// TIA Portal project "S7-1200-Tank-Level-Control" (V17)

(* hardware
DEVICE "S7-1200 station_1"  S7-1200 Station
   slot 0: "Rack_0"  S7-1200 Rack  Rack  V1.0
   slot 1: "PLC_1"  CPU 1212C DC/DC/DC  6ES7 212-1AE40-0XB0  V4.2
DEVICE "HMI_1"  TP700 Comfort
   slot 0: "HMI_1"  TP700 Comfort  6AV2 124-0GC01-0AX0  17.0.0.0
   slot 1: "HMI_RT_1"  TP700 Comfort  6AV2 124-0GC01-0AX0  17.0.0.0
   slot 5: "HMI_1.IE_CP_1"  PROFINET Interface  17.0.0.0
      slot 1: "PROFINET Interface_1"  PROFINET Interface
         slot 1: "Port_1"  Port
         slot 2: "Port_2"  Port
   slot 7: "HMI_1.MPI/DP_CP_1"  MPI/DP Interface  17.0.0.0
*)

// ===== PLC "PLC_1"  CPU 1212C DC/DC/DC =====

DATA_BLOCK "DB_Control"   // DB1
{ S7_Optimized_Access := 'TRUE' }
VERSION : 0.1
   VAR
      AutoMode : Bool;   // Automatic operating mode
      ManualInletCmd : Real;   // Manual inlet valve command [%]
      ManualOutletCmd : Real;   // Manual outlet valve command [%]
      PIDInletCmd : Real;   // PID controller output [%]
      InletValveCmd : Real;   // Final inlet valve command [%]
      OutletValveCmd : Real;   // Final outlet valve command [%]
      LevelSetpoint : Real := 50.0;   // Tank level setpoint [%]
      Level_H : Bool;   // High level alarm
      Level_HH : Bool;   // High-high level protection
      Level_L : Bool;   // Low level alarm
      Level_LL : Bool;   // Low-low level protection
      HMI_AlarmWord : Word;   // HMI alarm trigger word
      ManualPumpCmd : Bool;   // Manual pump command
      PumpManualControlEnable : Bool;   // Manual pump control permission
   END_VAR
BEGIN
END_DATA_BLOCK

DATA_BLOCK "DB_TankSimulation"   // DB2
{ S7_Optimized_Access := 'TRUE' }
VERSION : 0.1
// stored: InstanceOfName FB_TankSimulation
"FB_TankSimulation"
BEGIN
END_DATA_BLOCK

FUNCTION_BLOCK "FB_TankSimulation"   // FB1, SCL
{ S7_Optimized_Access := 'TRUE' }
VERSION : 0.1
   VAR_INPUT
      CycleTime : Real := 0.1;
      InletValveCmd : Real;
      OutletValveCmd : Real;
   END_VAR
   VAR
      TankLevel : Real;
      Inflow : Real;
      Outflow : Real;
      InletValveActual : Real;
      OutletValveActual : Real;
      ValveSpeed : Real := 5.0;
      PumpRunning : Bool;
      PumpSpeed : Real := 2.0;
      PumpTimer : Real;
      PumpFailureSimulation : Bool;
      PumpFault : Bool;
      PumpFaultReset : Bool;
      PumpCmd : Bool;
   END_VAR
BEGIN
   REGION Pump_simulation

       IF #PumpCmd AND NOT #PumpFault THEN
           #PumpTimer := #PumpTimer + (#PumpSpeed * #CycleTime);

           IF #PumpTimer >= 2.0 AND NOT #PumpFailureSimulation THEN
               #PumpRunning := TRUE;
               #PumpTimer := 2.0;

           ELSIF #PumpTimer >= 4.0 AND #PumpFailureSimulation THEN
               #PumpFault := TRUE;
               #PumpTimer := 0.0;
           END_IF;

       END_IF;

       IF NOT #PumpCmd THEN
           #PumpTimer := #PumpTimer - (#PumpSpeed * #CycleTime);

           IF #PumpTimer <= 0.0 THEN
               #PumpRunning := FALSE;
               #PumpTimer := 0.0;
           END_IF;

       END_IF;

       IF #PumpFailureSimulation AND #PumpRunning THEN
           #PumpRunning := FALSE;
           #PumpFault := TRUE;
           #PumpTimer := 0.0;
       END_IF;

       IF #PumpFaultReset AND NOT #PumpFailureSimulation THEN
           #PumpFault := FALSE;
       END_IF;

   END_REGION


   REGION Inlet_valve_simulation

       IF #InletValveActual < #InletValveCmd THEN
           #InletValveActual := #InletValveActual + (#ValveSpeed * #CycleTime);

           IF #InletValveActual > #InletValveCmd THEN
               #InletValveActual := #InletValveCmd;
           END_IF;

       ELSIF #InletValveActual > #InletValveCmd THEN
           #InletValveActual := #InletValveActual - (#ValveSpeed * #CycleTime);

           IF #InletValveActual < #InletValveCmd THEN
               #InletValveActual := #InletValveCmd;
           END_IF;

       END_IF;

   END_REGION


   REGION Outlet_valve_simulation

       IF #OutletValveActual < #OutletValveCmd THEN
           #OutletValveActual := #OutletValveActual + (#ValveSpeed * #CycleTime);

           IF #OutletValveActual > #OutletValveCmd THEN
               #OutletValveActual := #OutletValveCmd;
           END_IF;

       ELSIF #OutletValveActual > #OutletValveCmd THEN
           #OutletValveActual := #OutletValveActual - (#ValveSpeed * #CycleTime);

           IF #OutletValveActual < #OutletValveCmd THEN
               #OutletValveActual := #OutletValveCmd;
           END_IF;

       END_IF;

   END_REGION


   REGION Flow_calculation

       IF #PumpRunning THEN
           #Inflow := (#InletValveActual / 100.0) * 2.0;
       ELSE
           #Inflow := 0.0;
       END_IF;

       #Outflow := (#OutletValveActual / 100.0) * 2.0;

   END_REGION


   REGION Tank_level_simulation

       #TankLevel := #TankLevel + (#Inflow - #Outflow) * #CycleTime;

       IF #TankLevel > 100.0 THEN
           #TankLevel := 100.0;
       END_IF;

       IF #TankLevel < 0.0 THEN
           #TankLevel := 0.0;
       END_IF;

   END_REGION
END_FUNCTION_BLOCK

ORGANIZATION_BLOCK "Main"   // OB1, LAD, ProgramCycle
TITLE = "Main Program Sweep (Cycle)"
{ S7_Optimized_Access := 'TRUE' }
VERSION : 0.1
   VAR_INPUT
      Initial_Call : Bool;   // Initial call of this OB
      Remanence : Bool;   // =True, if remanent data are available
   END_VAR
BEGIN

REGION Network 1: Operating mode command selection
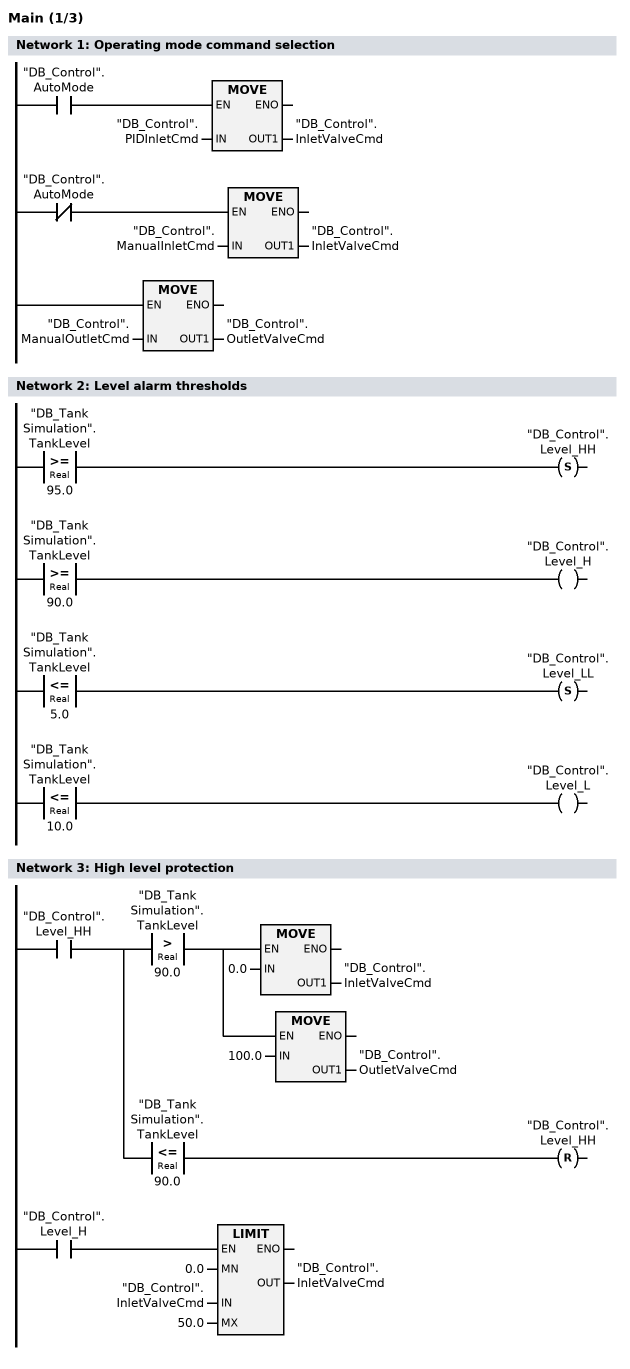
   RUNG wire#powerrail
      Contact( "DB_Control".AutoMode )
      Move(in := "DB_Control".PIDInletCmd, out1 => "DB_Control".InletValveCmd)
   END_RUNG
   RUNG wire#powerrail
      I_Contact( "DB_Control".AutoMode )
      Move(in := "DB_Control".ManualInletCmd, out1 => "DB_Control".InletValveCmd)
   END_RUNG
   RUNG wire#powerrail
      Move(in := "DB_Control".ManualOutletCmd, out1 => "DB_Control".OutletValveCmd)
   END_RUNG
   // the same network as SCL:
   IF "DB_Control".AutoMode THEN "DB_Control".InletValveCmd := "DB_Control".PIDInletCmd; END_IF;
   IF NOT "DB_Control".AutoMode THEN "DB_Control".InletValveCmd := "DB_Control".ManualInletCmd; END_IF;
   "DB_Control".OutletValveCmd := "DB_Control".ManualOutletCmd;
END_REGION

REGION Network 2: Level alarm thresholds
   RUNG wire#powerrail
      { S7_Templates := "SrcType := Real" } GE_Contact(in1 := "DB_TankSimulation".TankLevel, in2 := 95.0)
      S_Coil( "DB_Control".Level_HH )
   END_RUNG
   RUNG wire#powerrail
      { S7_Templates := "SrcType := Real" } GE_Contact(in1 := "DB_TankSimulation".TankLevel, in2 := 90.0)
      Coil( "DB_Control".Level_H )
   END_RUNG
   RUNG wire#powerrail
      { S7_Templates := "SrcType := Real" } LE_Contact(in1 := "DB_TankSimulation".TankLevel, in2 := 5.0)
      S_Coil( "DB_Control".Level_LL )
   END_RUNG
   RUNG wire#powerrail
      { S7_Templates := "SrcType := Real" } LE_Contact(in1 := "DB_TankSimulation".TankLevel, in2 := 10.0)
      Coil( "DB_Control".Level_L )
   END_RUNG
   // the same network as SCL:
   IF "DB_TankSimulation".TankLevel >= 95.0 THEN "DB_Control".Level_HH := TRUE; END_IF;
   "DB_Control".Level_H := "DB_TankSimulation".TankLevel >= 90.0;
   IF "DB_TankSimulation".TankLevel <= 5.0 THEN "DB_Control".Level_LL := TRUE; END_IF;
   "DB_Control".Level_L := "DB_TankSimulation".TankLevel <= 10.0;
END_REGION

REGION Network 3: High level protection
   IF "DB_Control".Level_HH AND ("DB_TankSimulation".TankLevel > 90.0) THEN
       "DB_Control".InletValveCmd := 0.0;
       "DB_Control".OutletValveCmd := 100.0;
   END_IF;
   IF "DB_Control".Level_HH AND ("DB_TankSimulation".TankLevel <= 90.0) THEN
       "DB_Control".Level_HH := FALSE;
   END_IF;
   IF "DB_Control".Level_H THEN
       "DB_Control".InletValveCmd := LIMIT(MN := 0.0, IN := "DB_Control".InletValveCmd, MX := 50.0);
   END_IF;
END_REGION

REGION Network 4: Low level protection
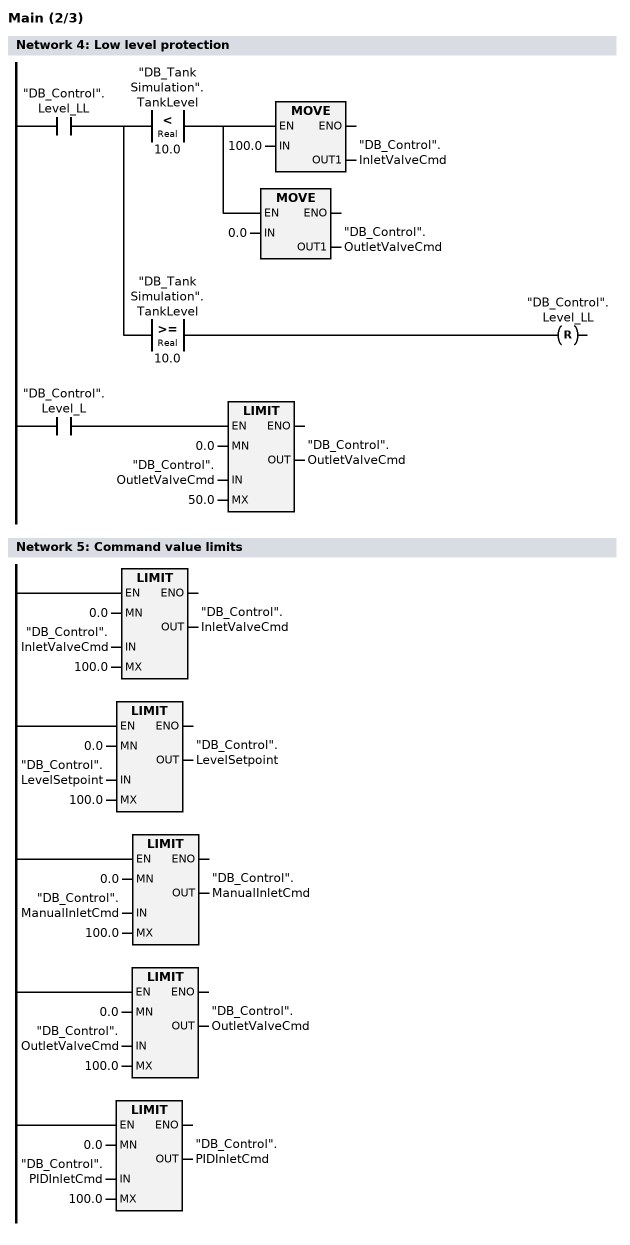
   IF "DB_Control".Level_LL AND ("DB_TankSimulation".TankLevel < 10.0) THEN
       "DB_Control".InletValveCmd := 100.0;
       "DB_Control".OutletValveCmd := 0.0;
   END_IF;
   IF "DB_Control".Level_LL AND ("DB_TankSimulation".TankLevel >= 10.0) THEN
       "DB_Control".Level_LL := FALSE;
   END_IF;
   IF "DB_Control".Level_L THEN
       "DB_Control".OutletValveCmd := LIMIT(MN := 0.0, IN := "DB_Control".OutletValveCmd, MX := 50.0);
   END_IF;
END_REGION

REGION Network 5: Command value limits
   "DB_Control".InletValveCmd := LIMIT(MN := 0.0, IN := "DB_Control".InletValveCmd, MX := 100.0);
   "DB_Control".LevelSetpoint := LIMIT(MN := 0.0, IN := "DB_Control".LevelSetpoint, MX := 100.0);
   "DB_Control".ManualInletCmd := LIMIT(MN := 0.0, IN := "DB_Control".ManualInletCmd, MX := 100.0);
   "DB_Control".OutletValveCmd := LIMIT(MN := 0.0, IN := "DB_Control".OutletValveCmd, MX := 100.0);
   "DB_Control".PIDInletCmd := LIMIT(MN := 0.0, IN := "DB_Control".PIDInletCmd, MX := 100.0);
END_REGION

REGION Network 6: HMI alarm word mapping
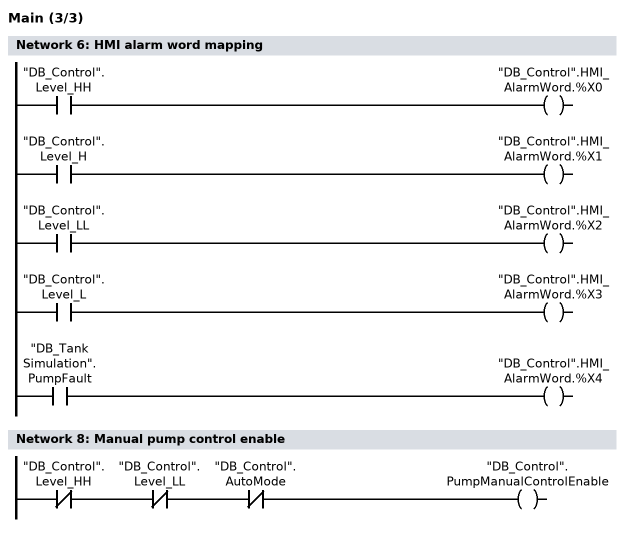
   RUNG wire#powerrail
      Contact( "DB_Control".Level_HH )
      Coil( "DB_Control".HMI_AlarmWord.%X0 )
   END_RUNG
   RUNG wire#powerrail
      Contact( "DB_Control".Level_H )
      Coil( "DB_Control".HMI_AlarmWord.%X1 )
   END_RUNG
   RUNG wire#powerrail
      Contact( "DB_Control".Level_LL )
      Coil( "DB_Control".HMI_AlarmWord.%X2 )
   END_RUNG
   RUNG wire#powerrail
      Contact( "DB_Control".Level_L )
      Coil( "DB_Control".HMI_AlarmWord.%X3 )
   END_RUNG
   RUNG wire#powerrail
      Contact( "DB_TankSimulation".PumpFault )
      Coil( "DB_Control".HMI_AlarmWord.%X4 )
   END_RUNG
   // the same network as SCL:
   "DB_Control".HMI_AlarmWord.%X0 := "DB_Control".Level_HH;
   "DB_Control".HMI_AlarmWord.%X1 := "DB_Control".Level_H;
   "DB_Control".HMI_AlarmWord.%X2 := "DB_Control".Level_LL;
   "DB_Control".HMI_AlarmWord.%X3 := "DB_Control".Level_L;
   "DB_Control".HMI_AlarmWord.%X4 := "DB_TankSimulation".PumpFault;
END_REGION

REGION Network 7 (SCL): Pump command control
   IF "DB_Control".Level_HH THEN
       "DB_TankSimulation".PumpCmd := FALSE;
   ELSIF "DB_Control".Level_LL THEN
       "DB_TankSimulation".PumpCmd := TRUE;
   ELSIF "DB_Control".AutoMode THEN
       "DB_TankSimulation".PumpCmd := TRUE;
   ELSE
       "DB_TankSimulation".PumpCmd := "DB_Control".ManualPumpCmd;

   END_IF;
END_REGION

REGION Network 8: Manual pump control enable
   RUNG wire#powerrail
      I_Contact( "DB_Control".Level_HH )
      I_Contact( "DB_Control".Level_LL )
      I_Contact( "DB_Control".AutoMode )
      Coil( "DB_Control".PumpManualControlEnable )
   END_RUNG
   // the same network as SCL:
   "DB_Control".PumpManualControlEnable := NOT "DB_Control".Level_HH AND NOT "DB_Control".Level_LL AND NOT "DB_Control".AutoMode;
END_REGION
END_ORGANIZATION_BLOCK

ORGANIZATION_BLOCK "OB_TankSimulation"   // OB30, LAD, CyclicInterrupt
{ S7_Optimized_Access := 'TRUE' }
VERSION : 0.1
   VAR_INPUT
      Initial_Call : Bool;   // Initial call of this OB
      Event_Count : Int;   // Events discarded
   END_VAR
BEGIN

REGION Network 1: Tank Simulation Execution
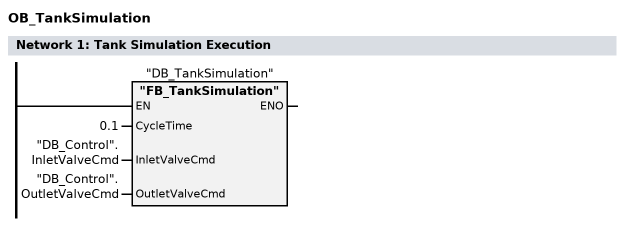
   RUNG wire#powerrail
      "DB_TankSimulation"(CycleTime := 0.1, InletValveCmd := "DB_Control".InletValveCmd, OutletValveCmd := "DB_Control".OutletValveCmd)
   END_RUNG
   // the same network as SCL:
   "DB_TankSimulation"(CycleTime := 0.1,   // "FB_TankSimulation"
                       InletValveCmd := "DB_Control".InletValveCmd,
                       OutletValveCmd := "DB_Control".OutletValveCmd);
END_REGION
END_ORGANIZATION_BLOCK

ORGANIZATION_BLOCK "OB_PID_Control"   // OB31, LAD, CyclicInterrupt
{ S7_Optimized_Access := 'TRUE' }
VERSION : 0.1
   VAR_INPUT
      Initial_Call : Bool;   // Initial call of this OB
      Event_Count : Int;   // Events discarded
   END_VAR
BEGIN

REGION Network 1: PID Controller Execution
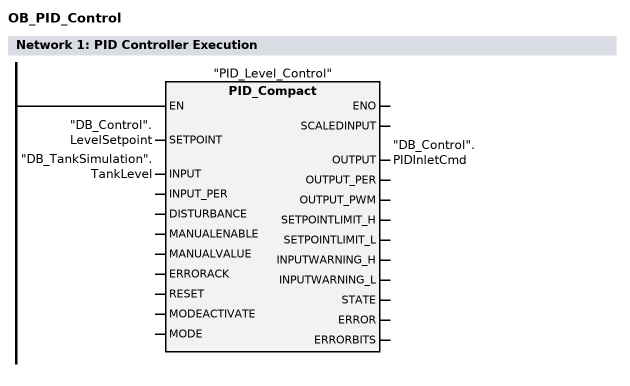
   "PID_Level_Control"(Setpoint := "DB_Control".LevelSetpoint,   // PID_Compact
                       Input := "DB_TankSimulation".TankLevel,
                       Output => "DB_Control".PIDInletCmd);
END_REGION
END_ORGANIZATION_BLOCK

(* ===== HMI "HMI_RT_1" =====
system functions are stored by id; their names below are inferred from use
connection "HMI_Connection_1": ETHERNET, S7_1200_OMS

HMI tags "Default tag table"
   "Tag_ScreenNumber" : UInt, internal
   "DB_Control_AutoMode" : Bool = PLC DB_Control.AutoMode, 1 s
   "DB_Control_LevelSetpoint" : Real = PLC DB_Control.LevelSetpoint, 1 s
   "DB_Control_ManualInletCmd" : Real = PLC DB_Control.ManualInletCmd, 1 s
   "DB_Control_OutletValveCmd" : Real = PLC DB_Control.OutletValveCmd, 1 s
   "DB_TankSimulation_TankLevel" : Real = PLC DB_TankSimulation.TankLevel, 1 s
   "DB_Control_PID_InletCmd" : Real = PLC DB_Control.PIDInletCmd, 1 s
   "DB_Control_InletValveCmd" : Real = PLC DB_Control.InletValveCmd, 1 s
   "DB_Control_Level_HH" : Bool = PLC DB_Control.Level_HH, 1 s
   "DB_Control_Level_H" : Bool = PLC DB_Control.Level_H, 1 s
   "DB_Control_Level_L" : Bool = PLC DB_Control.Level_L, 1 s
   "DB_Control_Level_LL" : Bool = PLC DB_Control.Level_LL, 1 s
   "DB_Control_ManualOutletCmd" : Real = PLC DB_Control.ManualOutletCmd, 1 s
   "DB_Control_HMI_AlarmWord" : Word = PLC DB_Control.HMI_AlarmWord, 1 s
   "DB_TankSimulation_OutletValveActual" : Real = PLC DB_TankSimulation.OutletValveActual, 1 s
   "DB_TankSimulation_InletValveActual" : Real = PLC DB_TankSimulation.InletValveActual, 1 s
   "DB_Control_ManualPumpCmd" : Bool = PLC DB_Control.ManualPumpCmd, 1 s
   "DB_TankSimulation_PumpRunning" : Bool = PLC DB_TankSimulation.PumpRunning, 1 s
   "DB_TankSimulation_PumpFault" : Bool = PLC DB_TankSimulation.PumpFault, 1 s
   "DB_TankSimulation_PumpFailureSimulation" : Bool = PLC DB_TankSimulation.PumpFailureSimulation, 1 s
   "DB_TankSimulation_PumpFaultReset" : Bool = PLC DB_TankSimulation.PumpFaultReset, 1 s
   "DB_Control_PumpManualControlEnable" : Bool = PLC DB_Control.PumpManualControlEnable, 1 s

discrete alarms
   1: 'Tank level above 95%', class Errors, trigger "DB_Control_HMI_AlarmWord" bit 0
   2: 'Tank level above 90%', class Warnings, trigger "DB_Control_HMI_AlarmWord" bit 1
   3: 'Tank level below 5%', class Errors, trigger "DB_Control_HMI_AlarmWord" bit 2
   4: 'Tank level below 10%', class Warnings, trigger "DB_Control_HMI_AlarmWord" bit 3
   5: 'Pump stopped', class Errors, trigger "DB_Control_HMI_AlarmWord" bit 4

screen "Tank Control" 800x428, template "Template_1"
   on GenerateScreen: SetTag("Tag_ScreenNumber", 1)
   TextField "Text field_1" at 89,0 size 149x23; Text 'CONTROL MODE'
   Circle "Circle_1" at 103,53 size 25x25
      Appearance <- "DB_Control_AutoMode"
   Circle "Circle_2" at 183,53 size 25x25
      Appearance <- "DB_Control_AutoMode"
   TextField "Text field_4" at 122,224 size 82x23; Text 'Setpoint'
   IOField "I/O field_1" at 128,247 size 67x32; FormatPattern 999
      ProcessValue <- "DB_Control_LevelSetpoint"
      ObjectEnable <- "DB_Control_AutoMode"
   TextField "Text field_5" at 163,251 size 25x23; Text '%'
   TextField "Text field_6" at 40,286 size 120x23; Text 'Manual Inlet'
   IOField "I/O field_2" at 62,308 size 67x32; FormatPattern 999
      ProcessValue <- "DB_Control_ManualInletCmd"
      ObjectEnable <- "DB_Control_AutoMode"
   TextField "Text field_7" at 97,312 size 25x23; Text '%'
   TextField "Text field_8" at 157,285 size 174x23; Text 'Outlet disturbance'
   IOField "I/O field_3" at 195,308 size 67x32; FormatPattern 999
      ProcessValue <- "DB_Control_ManualOutletCmd"
   TextField "Text field_9" at 230,312 size 25x23; Text '%'
   Bar "Bar_1" at 405,78 size 130x255; MinimumValue 0; MaximumValue 100
      ProcessValue <- "DB_TankSimulation_TankLevel"
   TextField "Text field_10" at 415,1 size 115x23; Text 'TANK LEVEL'
   IOField "I/O field_4" at 436,24 size 67x32; FormatPattern 999
      ProcessValue <- "DB_TankSimulation_TankLevel"
   TextField "Text field_11" at 471,28 size 25x23; Text '%'
   TextField "Text field_12" at 636,14 size 145x23; Text 'PROCESS DATA'
   TextField "Text field_13" at 611,47 size 82x23; Text 'Setpoint'
   IOField "I/O field_5" at 694,42 size 67x32; FormatPattern 999
      ProcessValue <- "DB_Control_LevelSetpoint"
   TextField "Text field_14" at 729,46 size 25x23; Text '%'
   TextField "Text field_15" at 611,85 size 104x23; Text 'Tank Level'
   IOField "I/O field_6" at 709,80 size 67x32; FormatPattern 999
      ProcessValue <- "DB_TankSimulation_TankLevel"
   TextField "Text field_16" at 744,84 size 25x23; Text '%'
   TextField "Text field_17" at 611,125 size 106x23; Text 'PID Output'
   IOField "I/O field_7" at 709,120 size 67x32; FormatPattern 999
      ProcessValue <- "DB_Control_PID_InletCmd"
   TextField "Text field_18" at 744,124 size 25x23; Text '%'
   TextField "Text field_19" at 612,163 size 103x23; Text 'Inlet valve'
   IOField "I/O field_8" at 709,159 size 67x32; FormatPattern 999
      ProcessValue <- "DB_TankSimulation_InletValveActual"
   TextField "Text field_20" at 744,163 size 25x23; Text '%'
   TextField "Text field_21" at 613,200 size 116x23; Text 'Outlet valve'
   IOField "I/O field_9" at 718,194 size 67x32; FormatPattern 999
      ProcessValue <- "DB_TankSimulation_OutletValveActual"
   TextField "Text field_22" at 753,198 size 25x23; Text '%'
   TextField "Text field_23" at 654,242 size 80x23; Text 'ALARMS'
   TextField "Text field_24" at 612,267 size 31x23; Text 'HH'
   TextField "Text field_25" at 709,267 size 18x23; Text 'H'
   TextField "Text field_26" at 612,310 size 25x23; Text 'LL'
   TextField "Text field_27" at 708,310 size 15x23; Text 'L'
   Circle "Circle_3" at 645,269 size 19x19
      Appearance <- "DB_Control_Level_HH"
   Circle "Circle_4" at 726,270 size 19x19
      Appearance <- "DB_Control_Level_H"
   Circle "Circle_5" at 645,312 size 19x19
      Appearance <- "DB_Control_Level_LL"
   Circle "Circle_6" at 726,312 size 19x19
      Appearance <- "DB_Control_Level_L"
   Button "Button_1" at 85,23 size 57x26; TextOff 'AUTO'
      on Press: SetBit("DB_Control_AutoMode")
   Button "Button_2" at 157,23 size 78x26; TextOff 'MANUAL'
      on Press: ResetBit("DB_Control_AutoMode")
   TextField "Text field_2" at 0,93 size 57x23; Text 'PUMP'
   Button "Button_3" at 59,88 size 69x31; TextOff 'START'
      on Press: SetBit("DB_Control_ManualPumpCmd")
      Visibility <- "DB_Control_ManualPumpCmd"
      ObjectEnable <- "DB_Control_PumpManualControlEnable"
   Button "Button_4" at 59,87 size 69x31; TextOff 'STOP'
      on Press: ResetBit("DB_Control_ManualPumpCmd")
      Visibility <- "DB_Control_ManualPumpCmd"
      ObjectEnable <- "DB_Control_PumpManualControlEnable"
   TextField "Text field_3" at 145,92 size 149x23; Text 'PUMP RUNNING'
   Circle "Circle_7" at 284,89 size 25x25
      Appearance <- "DB_TankSimulation_PumpRunning"
   Button "Button_5" at 3,143 size 169x32; TextOff 'FAULT SIMULATION'
      on Click: InvertBit("DB_TankSimulation_PumpFailureSimulation")
   TextField "Text field_28" at 91,186 size 137x23; Text 'FAULT ACTIVE'
   Circle "Circle_8" at 218,185 size 25x25
      Appearance <- "DB_TankSimulation_PumpFault"
   Button "Button_6" at 207,145 size 117x32; TextOff 'FAULT RESET'
      on Press: SetBit("DB_TankSimulation_PumpFaultReset")
      on Release: ResetBit("DB_TankSimulation_PumpFaultReset")

Template "Template_1" 800x428
   Button "Exit" at 720,360 size 78x58; TextOff 'Exit'; PictureOff "ExitRuntime_TP700_Comfort_TR"; PictureOn "ExitRuntime_TP700_Comfort_TR"
      on Release: StopRuntime(0)
   Button "Template_Button" at 640,360 size 78x58; TextOff 'Text'
   Button "Template_Button_1" at 560,360 size 78x58; TextOff 'Text'
   Button "Template_Button_2" at 480,360 size 78x58; TextOff 'Text'
   Button "Template_Button_3" at 400,360 size 78x58; TextOff 'Text'
   Button "Template_Button_4" at 321,360 size 78x58; TextOff 'Text'
   Button "Template_Button_5" at 241,360 size 78x58; TextOff 'Text'
   Button "Template_Button_6" at 161,360 size 78x58; TextOff 'Alarms'
      on Release: ActivateScreen("Alarms", 0)
   Button "Template_Button_7" at 81,360 size 78x58; TextOff 'Trends'
      on Release: ActivateScreen("Trends", 0)
   Button "Start screen" at 1,360 size 78x58; TextOff 'Start screen'; PictureOff "NavigateHome_TP700_Comfort_TR"; PictureOn "NavigateHome_TP700_Comfort_TR"
      on Release: ActivateScreen("Tank Control", 0)

screen "Trends" 800x428, template "Template_1"
   on GenerateScreen: SetTag("Tag_ScreenNumber", 2)
   TrendView "Trend view_1" at 0,0 size 799x359

screen "Alarms" 800x428, template "Template_1"
   on GenerateScreen: SetTag("Tag_ScreenNumber", 3)
   AlarmView "Alarm view_1" at 0,0 size 799x359
*)